Universal Robots PolyScope program: starting_point.urp

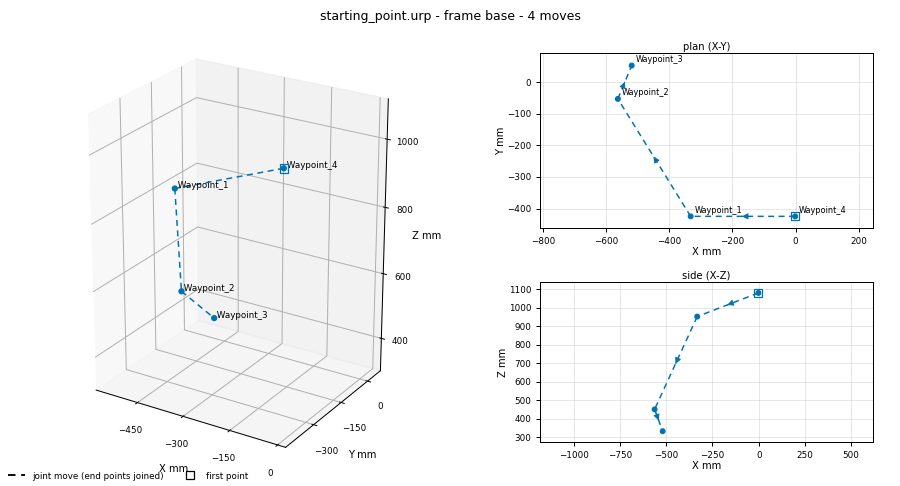
[picture p0: tool path of starting_point.urp in frame base, 4 of 4 moves have a stored position in this frame; points joined in program order, loops and branches not executed]
Program starting_point (installation=default directory=/programs/AronLauschOrdering createdIn=5.12.6.1102099 lastSavedIn=5.12.6.1102099 robotSerialNumber=20215500597)
Calibrated DH parameters: a=[0.000193, -0.066673, -0.391568, -0.000012, 0.00005, 0]; d=[0.162643, -472.05677, 465.132521, 7.058239, 0.099746, 0.099582]; alpha=[1.571116, 0.00089, 0.003862, 1.569269, -1.569248, 0]; deltaTheta=[0, -1.413394, 7.628392, 0.068187, 0, -0.000001]
Robot Program (runOnlyOnce=true)
  MoveJ speed 60 deg/s, acceleration 80 deg/s^2 (useActiveTCP=true) feature=Base
    Waypoint Waypoint_4: TCP in base x=-1.536 y=-424.817 z=1080.554 mm, rx=-0.0045 ry=-2.2186 rz=2.2204 rad; joints [0.001, -89.999, 0, -89.999, 0.002, 0.004] deg; TCP offset x=0 y=0 z=191.5 mm, rx=0 ry=0 rz=0 rad
    Waypoint Waypoint_1: TCP in base x=-332.388 y=-424.82 z=952.951 mm, rx=0.6923 ry=1.7965 rz=-1.7954 rad; joints [-0.004, -89.759, 41.77, -90.057, -0.006, 0.004] deg
    Waypoint Waypoint_2: TCP in base x=-562.913 y=-52.896 z=450.937 mm, rx=-2.3277 ry=-1.9474 rz=0.2663 rad; joints [-10.568, -87.01, 67.503, -81.011, -85.577, 0.009] deg
    Waypoint Waypoint_3: TCP in base x=-519.145 y=52.76 z=332.958 mm, rx=-3.1405 ry=-0.0837 rz=0.0002 rad; joints [-20.664, -88.123, 82.733, -84.528, -89.812, 66.326] deg
  URCap Gripper Activate (Robotiq_Grippers, Robotiq Inc.) dataModel(ResetAndActivateKey=false)
